TYPE E_DayPL :(Poniedzialek:=1, Wtorek, Sroda, Czwartek, Piatek, Sobota, Niedziela );
END_TYPE

(* stored: Version 1.1.0.1, ProductVersion 3.1.4019.2
   DUT E_DayPL: Id {215f77f9-b7bb-42a3-8014-21fc3529093e} *)
